TYPE ST_AteqIo :
STRUCT
	stIn  : ST_AteqInRead;
    stOut : ST_AteqOutWrite;
END_STRUCT
END_TYPE

(* stored: Version 1.1.0.1, ProductVersion 3.1.4024.15
   DUT ST_AteqIo: Id {7ce7ac0c-1c92-4cec-a3bd-bf1f5c9de48e} *)
